PROGRAM MAIN
VAR
	fbPlayList		: FB_SequenceManager;
	nTest			: INT;
END_VAR

IF (nTest = 1) THEN
	fbPlayList.Sort(E_SortedOrder.Id);
	nTest := 0;
ELSIF (nTest = 2) THEN
	fbPlayList.Sort(E_SortedOrder.Value);
	nTest := 0;
END_IF

END_PROGRAM

(* stored: Version 1.1.0.1, ProductVersion 3.1.4024.12
   POU MAIN: Id {79961382-ab79-4f28-a3a8-40d9a82cec0a}, SpecialFunc None *)
